FUNCTION_BLOCK Motor (* model behavior function block of DC Motor *)
  (* Standard: 61499-2 *)
  (* Version 1.0, 2018-02-26, Duc Do Tran, OFFIS e.V. *)
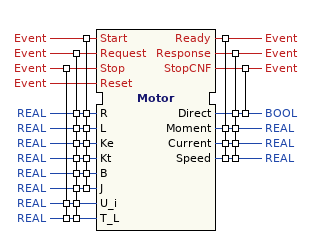
  EVENT_INPUT
    Start WITH R, L, Ke, J, B, Kt;
    Request WITH R, L, Ke, J, U_i, T_L, B, Kt;
    Stop WITH U_i, T_L;
    Reset;
  END_EVENT
  EVENT_OUTPUT
    Ready WITH Speed, Moment, Current;
    Response WITH Speed, Moment, Current, Direct;
    StopCNF WITH Direct;
  END_EVENT
  VAR_INPUT
    R : REAL := 2;
    L : REAL := 0.5;
    Ke : REAL := 0.1;
    Kt : REAL := 0.1;
    B : REAL := 0.2;
    J : REAL := 0.02;
    U_i : REAL;
    T_L : REAL;
  END_VAR
  VAR_OUTPUT
    Direct : BOOL;
    Moment : REAL;
    Current : REAL;
    Speed : REAL;
  END_VAR
  VAR
    deltaI : REAL := 0; (* Internal Variable *)
    t : REAL; (* Internal Variable *)
    bd : BOOL; (* Internal Variable *)
    deltaV : REAL; (* Internal Variable *)
    pi : REAL := 3.1415926; (* Internal Variable *)
    t0 : TIME; (* Internal Variable *)
    tg : TIME; (* Internal Variable *)
    omega : REAL; (* Internal Variable *)
  END_VAR
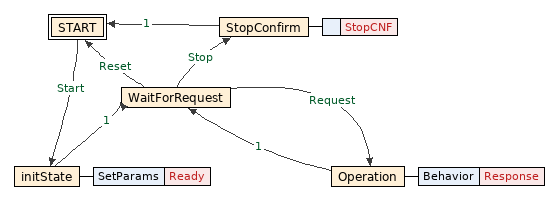
  EC_STATES
    START; (* Initial State *)
    initState : SetParams -> Ready;
    WaitForRequest;
    Operation : Behavior -> Response;
    StopConfirm : -> StopCNF;
  END_STATES
  EC_TRANSITIONS
    START TO initState := Start;
    initState TO WaitForRequest := 1;
    Operation TO WaitForRequest := 1;
    WaitForRequest TO Operation := Request;
    WaitForRequest TO StopConfirm := Stop;
    StopConfirm TO START := 1;
    WaitForRequest TO START := Reset;
  END_TRANSITIONS
  ALGORITHM SetParams IN ST: (* new algorithm *)
bd := TRUE;
Speed := 0;
Moment := 0;
Current := 0;
t := 0;
  END_ALGORITHM
  ALGORITHM Behavior IN ST: (* new algorithm *)
IF bd = TRUE THEN
	tg := NOW_MONOTONIC();
	bd := FALSE;
END_IF;
t := TIME_IN_S_TO_LREAL(NOW_MONOTONIC() - tg);
tg := NOW_MONOTONIC();
deltaI := (U_i - R*Current  - Ke* omega)*t/L;
Current :=Current + deltaI;
Moment := Kt*Current;
deltaV := (Moment - B*omega - T_L)*t/J;
omega := omega + deltaV;
Speed := omega;//
Direct := (U_i >= 0);
//Speed := omega*30/pi;
  END_ALGORITHM
END_FUNCTION_BLOCK
